Yaskawa INFORM job: kufsa_real.JBI

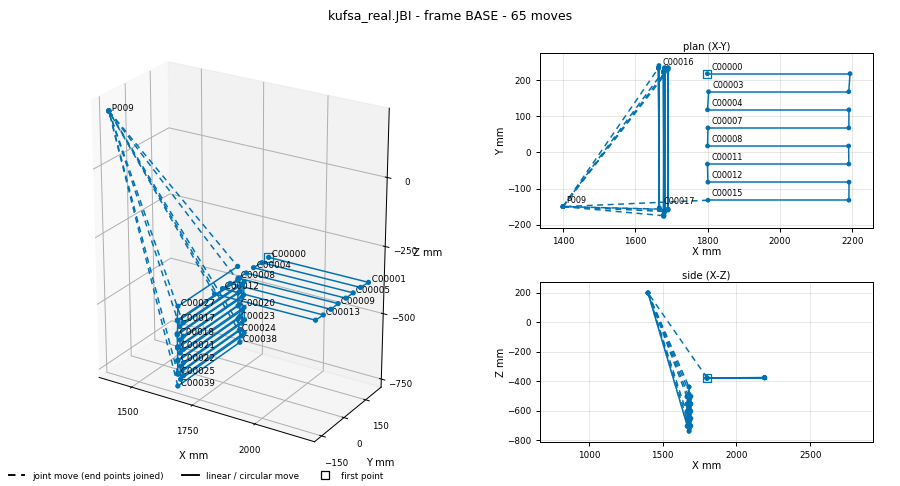
[picture p0: tool path of kufsa_real.JBI in frame BASE, 65 of 65 moves have a stored position in this frame; points joined in program order, loops and branches not executed]
/JOB
//NAME kufsa_real
//POS
///NPOS 60,0,60,1,0,0
///TOOL 0
///POSTYPE BASE
///RECTAN
///RCONF 1,0,0,0,0,0,0,0,0,0,0,0,0,0,0,0,0,0,0,0,0,0,0,0
C00000=1799.105,217.743,-376.719,180.0000,0.0000,0.0000
C00001=2193.209,217.743,-375.224,180.0000,0.0000,0.0000
C00002=2189.640,167.743,-375.035,180.0000,0.0000,0.0000
C00003=1802.416,167.743,-376.945,180.0000,0.0000,0.0000
C00004=1799.461,117.743,-377.155,180.0000,0.0000,0.0000
C00005=2190.175,117.743,-375.229,180.0000,0.0000,0.0000
C00006=2189.945,67.743,-374.707,180.0000,0.0000,0.0000
C00007=1800.555,67.743,-377.416,180.0000,0.0000,0.0000
C00008=1799.574,17.743,-377.432,180.0000,0.0000,0.0000
C00009=2189.258,17.743,-374.777,180.0000,0.0000,0.0000
C00010=2189.936,-32.256,-375.068,180.0000,0.0000,0.0000
C00011=1799.279,-32.256,-377.528,180.0000,0.0000,0.0000
C00012=1800.458,-82.256,-376.642,180.0000,0.0000,0.0000
C00013=2190.469,-82.256,-375.087,180.0000,0.0000,0.0000
C00014=2190.131,-132.256,-373.628,180.0000,0.0000,0.0000
C00015=1800.792,-132.256,-376.594,180.0000,0.0000,0.0000
C00016=1663.630,232.602,-503.508,180.0000,-89.9999,0.0000
C00017=1666.148,-152.983,-503.508,180.0000,-89.9999,0.0000
C00018=1666.041,-157.222,-553.508,180.0000,-89.9999,0.0000
C00019=1663.921,233.381,-553.508,180.0000,-89.9999,0.0000
C00020=1664.032,233.772,-603.508,180.0000,-89.9999,0.0000
C00021=1666.195,-156.635,-603.508,180.0000,-89.9999,0.0000
C00022=1666.144,-156.750,-653.508,180.0000,-89.9999,0.0000
C00023=1664.648,233.958,-653.508,180.0000,-89.9999,0.0000
C00024=1665.281,240.186,-703.508,180.0000,-89.9999,0.0000
C00025=1666.323,-156.758,-703.508,180.0000,-89.9999,0.0000
C00026=1677.678,209.846,-437.485,180.0000,-89.9999,0.0000
C00027=1678.733,-170.147,-437.485,180.0000,-89.9999,0.0000
C00028=1678.640,-174.851,-487.485,180.0000,-89.9999,0.0000
C00029=1677.720,223.186,-487.485,180.0000,-89.9999,0.0000
C00030=1679.116,221.336,-537.485,180.0000,-89.9999,0.0000
C00031=1678.510,-176.882,-537.485,180.0000,-89.9999,0.0000
C00032=1678.539,-175.322,-587.485,180.0000,-89.9999,0.0000
C00033=1678.922,222.387,-587.485,180.0000,-89.9999,0.0000
C00034=1677.674,223.803,-637.485,180.0000,-89.9999,0.0000
C00035=1678.841,-175.651,-637.485,180.0000,-89.9999,0.0000
C00036=1678.086,-175.495,-687.485,180.0000,-89.9999,0.0000
C00037=1678.879,222.804,-687.485,180.0000,-89.9999,0.0000
C00038=1679.569,221.289,-737.485,180.0000,-89.9999,0.0000
C00039=1677.443,-175.016,-737.485,180.0000,-89.9999,0.0000
C00040=1690.476,-158.083,-501.808,180.0000,-89.9999,0.0000
C00041=1690.334,232.310,-501.808,180.0000,-89.9999,0.0000
C00042=1690.515,228.872,-551.808,180.0000,-89.9999,0.0000
C00043=1690.213,-157.792,-551.808,180.0000,-89.9999,0.0000
C00044=1689.886,-159.444,-601.808,180.0000,-89.9999,0.0000
C00045=1690.200,231.911,-601.808,180.0000,-89.9999,0.0000
C00046=1690.555,234.541,-651.808,180.0000,-89.9999,0.0000
C00047=1690.322,-157.870,-651.808,180.0000,-89.9999,0.0000
C00048=1689.273,-157.628,-701.808,180.0000,-89.9999,0.0000
C00049=1690.491,232.591,-701.808,180.0000,-89.9999,0.0000
C00050=1680.766,-163.387,-515.527,180.0000,-89.9999,0.0000
C00051=1680.834,234.142,-515.527,180.0000,-89.9999,0.0000
C00052=1680.687,233.311,-565.527,180.0000,-89.9999,0.0000
C00053=1681.066,-163.618,-565.527,180.0000,-89.9999,0.0000
C00054=1681.334,-163.573,-615.527,180.0000,-89.9999,0.0000
C00055=1681.446,233.261,-615.527,180.0000,-89.9999,0.0000
C00056=1681.738,230.395,-665.527,180.0000,-89.9999,0.0000
C00057=1681.212,-162.975,-665.527,180.0000,-89.9999,0.0000
C00058=1681.395,-163.194,-715.527,180.0000,-89.9999,0.0000
C00059=1681.907,230.406,-715.527,180.0000,-89.9999,0.0000
///POSTYPE PULSE
///PULSE
EC00000=0
EC00001=0
EC00002=0
EC00003=0
EC00004=0
EC00005=0
EC00006=0
EC00007=0
EC00008=0
EC00009=0
EC00010=0
EC00011=0
EC00012=0
EC00013=0
EC00014=0
EC00015=0
EC00016=0
EC00017=0
EC00018=0
EC00019=0
EC00020=0
EC00021=0
EC00022=0
EC00023=0
EC00024=0
EC00025=0
EC00026=92160
EC00027=92160
EC00028=92160
EC00029=92160
EC00030=92160
EC00031=92160
EC00032=92160
EC00033=92160
EC00034=92160
EC00035=92160
EC00036=92160
EC00037=92160
EC00038=92160
EC00039=92160
EC00040=184320
EC00041=184320
EC00042=184320
EC00043=184320
EC00044=184320
EC00045=184320
EC00046=184320
EC00047=184320
EC00048=184320
EC00049=184320
EC00050=276480
EC00051=276480
EC00052=276480
EC00053=276480
EC00054=276480
EC00055=276480
EC00056=276480
EC00057=276480
EC00058=276480
EC00059=276480
///POSTYPE BASE
///RECTAN
P00009=1399.998,-150.003,199.998,-135.0004,-0.0006,-89.9996
//INST
///DATE 2023/01/17 15:33
///ATTR SC,RW,RJ
////FRAME BASE
///GROUP1 RB1,ST1
NOP
MOVJ C00000 EC00000 VJ=15.00
CALL JOB:SPYON
MOVL C00001 EC00001 V=200.0
MOVL C00002 EC00002 V=200.0
MOVL C00003 EC00003 V=200.0
MOVL C00004 EC00004 V=200.0
MOVL C00005 EC00005 V=200.0
MOVL C00006 EC00006 V=200.0
MOVL C00007 EC00007 V=200.0
MOVL C00008 EC00008 V=200.0
MOVL C00009 EC00009 V=200.0
MOVL C00010 EC00010 V=200.0
MOVL C00011 EC00011 V=200.0
MOVL C00012 EC00012 V=200.0
MOVL C00013 EC00013 V=200.0
MOVL C00014 EC00014 V=200.0
MOVL C00015 EC00015 V=200.0
CALL JOB:SPYOF
MOVJ P009 VJ=15.00
MOVJ C00016 EC00016 VJ=15.00
CALL JOB:SPYON
MOVL C00017 EC00017 V=200.0
MOVL C00018 EC00018 V=200.0
MOVL C00019 EC00019 V=200.0
MOVL C00020 EC00020 V=200.0
MOVL C00021 EC00021 V=200.0
MOVL C00022 EC00022 V=200.0
MOVL C00023 EC00023 V=200.0
MOVL C00024 EC00024 V=200.0
MOVL C00025 EC00025 V=200.0
CALL JOB:SPYOF
MOVJ P009 VJ=15.00
MOVJ C00026 EC00026 VJ=15.00
CALL JOB:SPYON
MOVL C00027 EC00027 V=200.0
MOVL C00028 EC00028 V=200.0
MOVL C00029 EC00029 V=200.0
MOVL C00030 EC00030 V=200.0
MOVL C00031 EC00031 V=200.0
MOVL C00032 EC00032 V=200.0
MOVL C00033 EC00033 V=200.0
MOVL C00034 EC00034 V=200.0
MOVL C00035 EC00035 V=200.0
MOVL C00036 EC00036 V=200.0
MOVL C00037 EC00037 V=200.0
MOVL C00038 EC00038 V=200.0
MOVL C00039 EC00039 V=200.0
CALL JOB:SPYOF
MOVJ P009 VJ=15.00
MOVJ C00040 EC00040 VJ=15.00
CALL JOB:SPYON
MOVL C00041 EC00041 V=200.0
MOVL C00042 EC00042 V=200.0
MOVL C00043 EC00043 V=200.0
MOVL C00044 EC00044 V=200.0
MOVL C00045 EC00045 V=200.0
MOVL C00046 EC00046 V=200.0
MOVL C00047 EC00047 V=200.0
MOVL C00048 EC00048 V=200.0
MOVL C00049 EC00049 V=200.0
CALL JOB:SPYOF
MOVJ P009 VJ=15.00
MOVJ C00050 EC00050 VJ=15.00
CALL JOB:SPYON
MOVL C00051 EC00051 V=200.0
MOVL C00052 EC00052 V=200.0
MOVL C00053 EC00053 V=200.0
MOVL C00054 EC00054 V=200.0
MOVL C00055 EC00055 V=200.0
MOVL C00056 EC00056 V=200.0
MOVL C00057 EC00057 V=200.0
MOVL C00058 EC00058 V=200.0
MOVL C00059 EC00059 V=200.0
CALL JOB:SPYOF
MOVJ P009 VJ=15.00
END
